// TIA Portal project "FinalPLC_V17" (V17)

(* hardware
DEVICE "S7-1200 station_1"  S7-1200 Station
   slot 0: "Rack_0"  S7-1200 Rack  Rack  V1.0
   slot 1: "PLC_1"  CPU 1211C DC/DC/DC  6ES7 211-1AE40-0XB0  V4.2
*)

// ===== PLC "PLC_1"  CPU 1211C DC/DC/DC =====

VAR_GLOBAL   // PLC tag table "Default tag table"
   "START" AT %I0.1 : Bool;
   "TG1" AT %M0.0 : Bool;
   "TG4" AT %M0.1 : Bool;
   "STOP" AT %I0.3 : Bool;
   "Emergency stop" AT %I0.4 : Bool;
   "AUTO" AT %I0.5 : Bool;
   "TG3" AT %M1.1 : Bool;
   "Entry Converyor" AT %Q0.0 : Bool;
   "Exit Converyor" AT %Q0.2 : Bool;
   "Start Light" AT %Q1.1 : Bool;
   "Start Light (Green)" AT %Q3.1 : Bool;
   "Stop Light (Red)" AT %Q3.3 : Bool;
   "Sensor 1" AT %I0.6 : Bool;
   "Vision sensor" AT %I0.0 : Bool;
   "Sensor 4" AT %I0.7 : Bool;
   "Output Vision" AT %ID30 : DInt;
   "Sortter 1 Turn" AT %Q0.3 : Bool;
   "TG STOP CG" AT %M0.2 : Bool;
   "Sortter 1 Belt" AT %Q0.4 : Bool;
   "RESET" AT %I0.2 : Bool;
   "Counter 1" AT %QD30 : DInt;
   "Sotter 2 Turn" AT %Q0.5 : Bool;
   "Sortter 2 Belt" AT %Q0.6 : Bool;
   "Counter 2" AT %QD34 : DInt;
   "Sotter 3 Turn" AT %Q0.7 : Bool;
   "Sotter 3 Belt" AT %Q1.0 : Bool;
   "Counter 3" AT %QD38 : DInt;
   "Counter 4" AT %QD42 : DInt;
   "TG5" AT %M0.5 : Bool;
   "Reset Light" AT %Q1.2 : Bool;
   "Reset Light (Yellow)" AT %Q3.2 : Bool;
   "Alarm Siren" AT %Q0.1 : Bool;
   "TG6" AT %M0.3 : Bool;
   "Grab 1" AT %Q2.3 : Bool;
   "Tag_1" AT %M100.0 : Bool;
   "Belt Converyor 1" AT %Q1.4 : Bool;
   "Belt Converyor 2" AT %Q1.5 : Bool;
   "Clamp 1" AT %Q1.7 : Bool;
   "Raise 1" AT %Q2.0 : Bool;
   "Sensor 3" AT %I1.1 : Bool;
   "Tag_2" AT %M100.1 : Bool;
   "Clamped 1" AT %I1.3 : Bool;
   "Mover Z1" AT %Q2.1 : Bool;
   "Detected 1" AT %I1.5 : Bool;
   "CB Sensor4" AT %M100.3 : Bool;
   "Moving Z1" AT %I1.6 : Bool;
   "Tag_10" AT %M101.1 : Bool;
   "Tag_3" AT %M100.2 : Bool;
   "Mover X1" AT %Q2.2 : Bool;
   "Clamp 2" AT %Q2.4 : Bool;
   "Clamped 2" AT %I2.0 : Bool;
   "Tag_5" AT %M100.4 : Bool;
   "Tag_6" AT %M100.5 : Bool;
   "Tag_8" AT %M100.7 : Bool;
   "Raise 2" AT %Q2.5 : Bool;
   "Tag_7" AT %M100.6 : Bool;
   "Sensor 2" AT %I1.0 : Bool;
   "Sensor box" AT %I1.2 : Bool;
   "Box converyor" AT %Q1.6 : Bool;
   "Tag_11" AT %M200.0 : Bool;
   "Mover Z2" AT %Q2.6 : Bool;
   "Mover X2" AT %Q2.7 : Bool;
   "Moving X2" AT %I2.4 : Bool;
   "Tag_12" AT %M200.1 : Bool;
   "Moving Z2" AT %I2.3 : Bool;
   "Tag_13" AT %M200.2 : Bool;
   "Grab 2" AT %Q3.0 : Bool;
   "Detected 2" AT %I2.2 : Bool;
   "Tag_14" AT %M200.3 : Bool;
   "Tag_15" AT %M200.4 : Bool;
   "Tag_19" AT %M200.7 : Bool;
   "Tag_16" AT %M200.5 : Bool;
   "Stop Light" AT %Q1.3 : Bool;
   "Tag_17" AT %M200.6 : Bool;
   "Tag_18" AT %QD46 : DInt;
   "Moving X1" AT %I1.7 : Bool;
   "Limit 1" AT %I1.4 : Bool;
   "TG2" AT %M1.0 : Bool;
   "MAN" AT %I2.5 : Bool;
   "IM_Con1" AT %I2.6 : Bool;
   "IM_Con2" AT %I2.7 : Bool;
   "IM_Con3" AT %I3.0 : Bool;
   "IM_Con4" AT %I3.1 : Bool;
   "IM_Alarm" AT %I3.2 : Bool;
END_VAR

// folder: System blocks/Program resources

DATA_BLOCK "IEC_Counter_0_DB"   // DB1
{ S7_Optimized_Access := 'TRUE' }
AUTHOR : SIMATIC
FAMILY : IEC
NAME : DCNTR
VERSION : 1.2
// stored: InstanceOfName IEC_DCOUNTER
"IEC_DCOUNTER"
BEGIN
END_DATA_BLOCK

DATA_BLOCK "IEC_Counter_0_DB_1"   // DB2
{ S7_Optimized_Access := 'TRUE' }
AUTHOR : SIMATIC
FAMILY : IEC
NAME : DCNTR
VERSION : 1.2
// stored: InstanceOfName IEC_DCOUNTER
"IEC_DCOUNTER"
BEGIN
END_DATA_BLOCK

DATA_BLOCK "IEC_Counter_0_DB_2"   // DB3
{ S7_Optimized_Access := 'TRUE' }
AUTHOR : SIMATIC
FAMILY : IEC
NAME : DCNTR
VERSION : 1.2
// stored: InstanceOfName IEC_DCOUNTER
"IEC_DCOUNTER"
BEGIN
END_DATA_BLOCK

DATA_BLOCK "IEC_Counter_0_DB_3"   // DB4
{ S7_Optimized_Access := 'TRUE' }
AUTHOR : SIMATIC
FAMILY : IEC
NAME : DCNTR
VERSION : 1.2
// stored: InstanceOfName IEC_DCOUNTER
"IEC_DCOUNTER"
BEGIN
END_DATA_BLOCK

DATA_BLOCK "IEC_Timer_0_DB"   // DB5
{ S7_Optimized_Access := 'TRUE' }
AUTHOR : Simatic
FAMILY : IEC
NAME : IEC_TMR
VERSION : 1.0
// stored: InstanceOfName IEC_TIMER
"IEC_TIMER"
BEGIN
END_DATA_BLOCK

DATA_BLOCK "IEC_Timer_0_DB_1"   // DB6
{ S7_Optimized_Access := 'TRUE' }
AUTHOR : Simatic
FAMILY : IEC
NAME : IEC_TMR
VERSION : 1.0
// stored: InstanceOfName IEC_TIMER
"IEC_TIMER"
BEGIN
END_DATA_BLOCK

DATA_BLOCK "IEC_Timer_0_DB_2"   // DB7
{ S7_Optimized_Access := 'TRUE' }
AUTHOR : Simatic
FAMILY : IEC
NAME : IEC_TMR
VERSION : 1.0
// stored: InstanceOfName IEC_TIMER
"IEC_TIMER"
BEGIN
END_DATA_BLOCK

DATA_BLOCK "IEC_Timer_0_DB_3"   // DB8
{ S7_Optimized_Access := 'TRUE' }
AUTHOR : Simatic
FAMILY : IEC
NAME : IEC_TMR
VERSION : 1.0
// stored: InstanceOfName IEC_TIMER
"IEC_TIMER"
BEGIN
END_DATA_BLOCK

DATA_BLOCK "IEC_Timer_0_DB_4"   // DB9
{ S7_Optimized_Access := 'TRUE' }
AUTHOR : Simatic
FAMILY : IEC
NAME : IEC_TMR
VERSION : 1.0
// stored: InstanceOfName IEC_TIMER
"IEC_TIMER"
BEGIN
END_DATA_BLOCK

DATA_BLOCK "IEC_Timer_0_DB_5"   // DB10
{ S7_Optimized_Access := 'TRUE' }
AUTHOR : Simatic
FAMILY : IEC
NAME : IEC_TMR
VERSION : 1.0
// stored: InstanceOfName IEC_TIMER
"IEC_TIMER"
BEGIN
END_DATA_BLOCK

DATA_BLOCK "IEC_Timer_0_DB_6"   // DB11
{ S7_Optimized_Access := 'TRUE' }
AUTHOR : Simatic
FAMILY : IEC
NAME : IEC_TMR
VERSION : 1.0
// stored: InstanceOfName IEC_TIMER
"IEC_TIMER"
BEGIN
END_DATA_BLOCK

DATA_BLOCK "IEC_Counter_0_DB_4"   // DB12
{ S7_Optimized_Access := 'TRUE' }
AUTHOR : SIMATIC
FAMILY : IEC
NAME : DCNTR
VERSION : 1.2
// stored: InstanceOfName IEC_DCOUNTER
"IEC_DCOUNTER"
BEGIN
END_DATA_BLOCK

// folder: (top level)

FUNCTION "Sorting station" : Void   // FC1, LAD
{ S7_Optimized_Access := 'TRUE' }
VERSION : 0.1
   VAR_TEMP   // added for the SCL form of the ladder/FBD networks
      _w1 : Bool;
   END_VAR
BEGIN

REGION Network 1: CHUONG TRINH
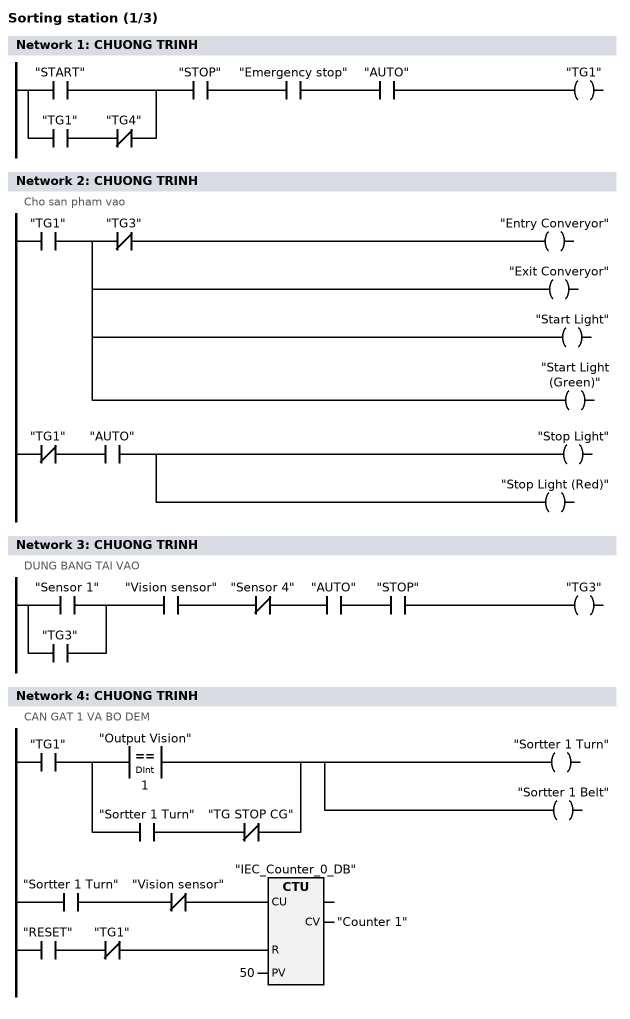
   RUNG wire#powerrail
      Contact( "START" )
      wire#w1
      Contact( "STOP" )
      Contact( "Emergency stop" )
      Contact( "AUTO" )
      Coil( "TG1" )
   END_RUNG
   RUNG wire#powerrail
      Contact( "TG1" )
      I_Contact( "TG4" )
   END_RUNG wire#w1
   // the same network as SCL:
   "TG1" := ("START" OR ("TG1" AND NOT "TG4")) AND "STOP" AND "Emergency stop" AND "AUTO";
END_REGION

REGION Network 2: CHUONG TRINH
   // Cho san pham vao
   RUNG wire#powerrail
      Contact( "TG1" )
      wire#w1
      I_Contact( "TG3" )
      Coil( "Entry Converyor" )
   END_RUNG
   RUNG wire#w1
      Coil( "Exit Converyor" )
   END_RUNG
   RUNG wire#w1
      Coil( "Start Light" )
   END_RUNG
   RUNG wire#w1
      Coil( "Start Light (Green)" )
   END_RUNG
   RUNG wire#powerrail
      I_Contact( "TG1" )
      Contact( "AUTO" )
      wire#w2
      Coil( "Stop Light" )
   END_RUNG
   RUNG wire#w2
      Coil( "Stop Light (Red)" )
   END_RUNG
   // the same network as SCL:
   "Entry Converyor" := "TG1" AND NOT "TG3";
   "Exit Converyor" := "TG1";
   "Start Light" := "TG1";
   "Start Light (Green)" := "TG1";
   "Stop Light" := NOT "TG1" AND "AUTO";
   "Stop Light (Red)" := "Stop Light";
END_REGION

REGION Network 3: CHUONG TRINH
   // DUNG BANG TAI VAO
   RUNG wire#powerrail
      Contact( "Sensor 1" )
      wire#w1
      Contact( "Vision sensor" )
      I_Contact( "Sensor 4" )
      Contact( "AUTO" )
      Contact( "STOP" )
      Coil( "TG3" )
   END_RUNG
   RUNG wire#powerrail
      Contact( "TG3" )
   END_RUNG wire#w1
   // the same network as SCL:
   "TG3" := ("Sensor 1" OR "TG3") AND "Vision sensor" AND NOT "Sensor 4" AND "AUTO" AND "STOP";
END_REGION

REGION Network 4: CHUONG TRINH
   // CAN GAT 1 VA BO DEM
   "Sortter 1 Turn" := "TG1" AND (("Output Vision" = 1) OR ("Sortter 1 Turn" AND NOT "TG STOP CG"));
   "Sortter 1 Belt" := "Sortter 1 Turn";
   "IEC_Counter_0_DB".CTU(CU := "Sortter 1 Turn" AND NOT "Vision sensor",
                          R := "RESET" AND NOT "TG1",
                          PV := 50,
                          CV => "Counter 1");
END_REGION

REGION Network 5: CHUONG TRINH
   // CAN GAT 2 VA BO DEM
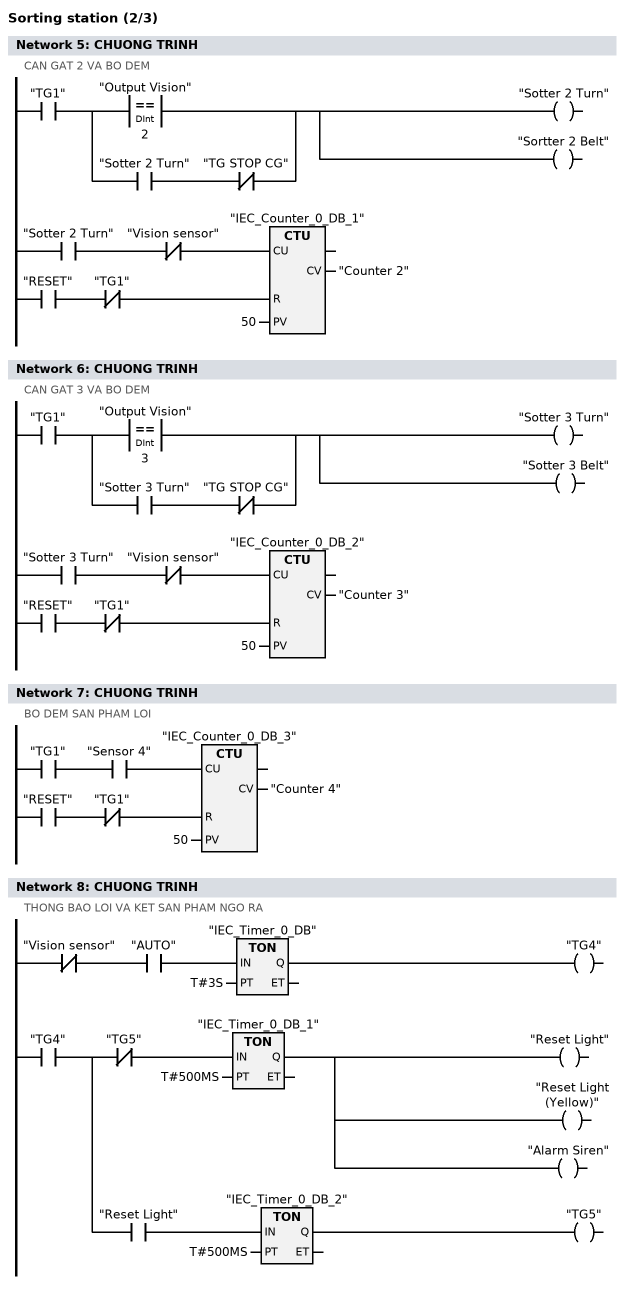
   "Sotter 2 Turn" := "TG1" AND (("Output Vision" = 2) OR ("Sotter 2 Turn" AND NOT "TG STOP CG"));
   "Sortter 2 Belt" := "Sotter 2 Turn";
   "IEC_Counter_0_DB_1".CTU(CU := "Sotter 2 Turn" AND NOT "Vision sensor",
                           R := "RESET" AND NOT "TG1",
                           PV := 50,
                           CV => "Counter 2");
END_REGION

REGION Network 6: CHUONG TRINH
   // CAN GAT 3 VA BO DEM
   "Sotter 3 Turn" := "TG1" AND (("Output Vision" = 3) OR ("Sotter 3 Turn" AND NOT "TG STOP CG"));
   "Sotter 3 Belt" := "Sotter 3 Turn";
   "IEC_Counter_0_DB_2".CTU(CU := "Sotter 3 Turn" AND NOT "Vision sensor",
                           R := "RESET" AND NOT "TG1",
                           PV := 50,
                           CV => "Counter 3");
END_REGION

REGION Network 7: CHUONG TRINH
   // BO DEM SAN PHAM LOI
   "IEC_Counter_0_DB_3".CTU(CU := "TG1" AND "Sensor 4", R := "RESET" AND NOT "TG1", PV := 50, CV => "Counter 4");
END_REGION

REGION Network 8: CHUONG TRINH
   // THONG BAO LOI VA KET SAN PHAM NGO RA
   "IEC_Timer_0_DB".TON(IN := NOT "Vision sensor" AND "AUTO", PT := T#3S);
   "TG4" := "IEC_Timer_0_DB".Q;
   "IEC_Timer_0_DB_1".TON(IN := "TG4" AND NOT "TG5", PT := T#500MS);
   "Reset Light" := "IEC_Timer_0_DB_1".Q;
   "Reset Light (Yellow)" := "IEC_Timer_0_DB_1".Q;
   "Alarm Siren" := "IEC_Timer_0_DB_1".Q;
   "IEC_Timer_0_DB_2".TON(IN := "TG4" AND "Reset Light", PT := T#500MS);
   "TG5" := "IEC_Timer_0_DB_2".Q;
END_REGION

REGION Network 9: CHUONG TRINH
   // THOI GIAN DELAY 1S CHO CAC CAN GAT
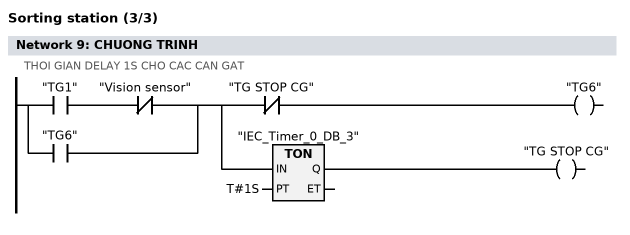
   #_w1 := ("TG1" AND NOT "Vision sensor") OR "TG6";
   "TG6" := #_w1 AND NOT "TG STOP CG";
   "IEC_Timer_0_DB_3".TON(IN := #_w1, PT := T#1S);
   "TG STOP CG" := "IEC_Timer_0_DB_3".Q;
END_REGION
END_FUNCTION

FUNCTION "Pick & Place 1" : Void   // FC2, LAD
{ S7_Optimized_Access := 'TRUE' }
VERSION : 0.1
   VAR_TEMP   // added for the SCL form of the ladder/FBD networks
      _w1 : Bool;
      _w2 : Bool;
      _w3 : Bool;
      _w4 : Bool;
      _w5 : Bool;
      _w6 : Bool;
   END_VAR
BEGIN

REGION Network 1
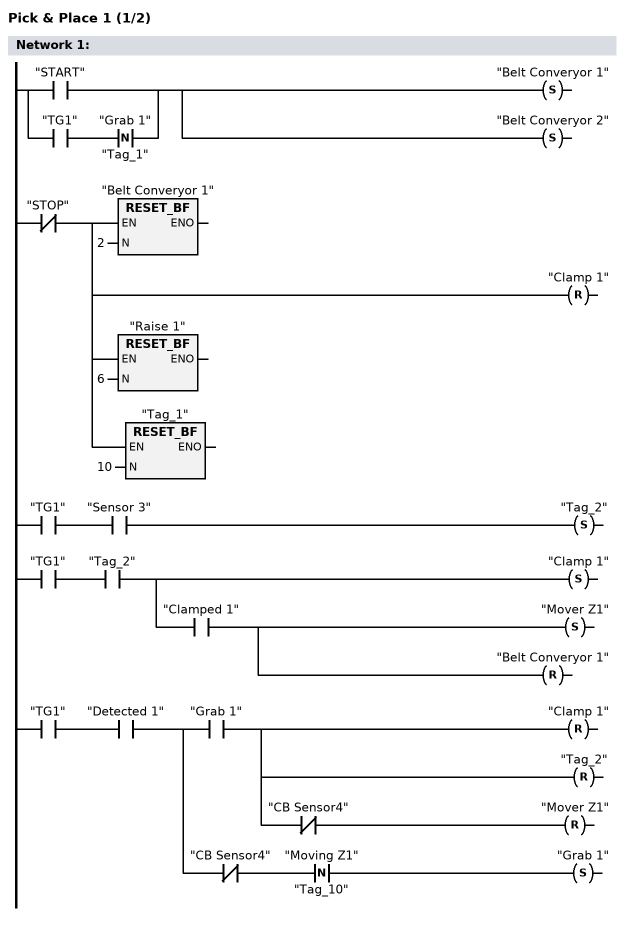
   // no SCL statement known for RBitfield: written as a call
   #_w1 := "TG1" AND NOT "Grab 1" AND "Tag_1";   // falling edge of "Grab 1"
   "Tag_1" := "Grab 1";
   IF "START" OR #_w1 THEN
       "Belt Converyor 1" := TRUE;
       "Belt Converyor 2" := TRUE;
   END_IF;
   #_w2 := NOT "STOP";
   IF #_w2 THEN
       RESET_BF(operand := "Belt Converyor 1", n := 2);
       "Clamp 1" := FALSE;
       RESET_BF(operand := "Raise 1", n := 6);
       RESET_BF(operand := "Tag_1", n := 10);
   END_IF;
   IF "TG1" AND "Sensor 3" THEN "Tag_2" := TRUE; END_IF;
   #_w3 := "TG1" AND "Tag_2";
   IF #_w3 THEN "Clamp 1" := TRUE; END_IF;
   IF #_w3 AND "Clamped 1" THEN
       "Mover Z1" := TRUE;
       "Belt Converyor 1" := FALSE;
   END_IF;
   #_w4 := "TG1" AND "Detected 1";
   #_w5 := #_w4 AND "Grab 1";
   IF #_w5 THEN
       "Clamp 1" := FALSE;
       "Tag_2" := FALSE;
   END_IF;
   IF #_w5 AND NOT "CB Sensor4" THEN "Mover Z1" := FALSE; END_IF;
   #_w6 := #_w4 AND NOT "CB Sensor4" AND NOT "Moving Z1" AND "Tag_10";   // falling edge of "Moving Z1"
   "Tag_10" := "Moving Z1";
   IF #_w6 THEN "Grab 1" := TRUE; END_IF;
END_REGION

REGION Network 2
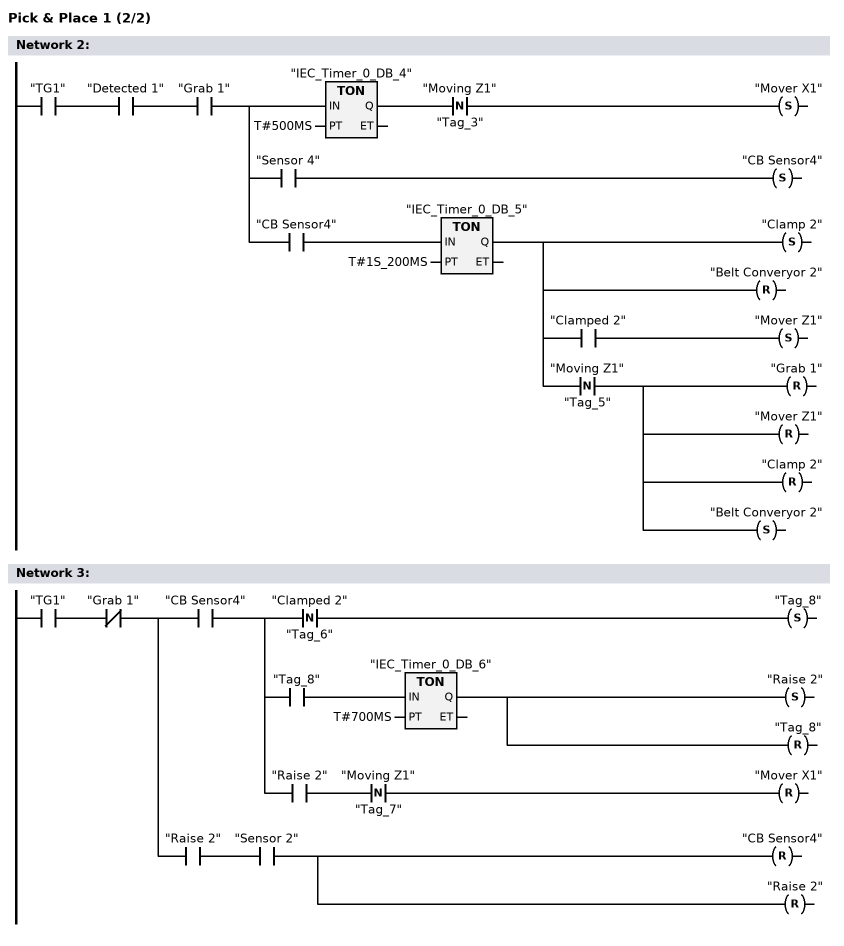
   #_w1 := "TG1" AND "Detected 1" AND "Grab 1";
   "IEC_Timer_0_DB_4".TON(IN := #_w1, PT := T#500MS);
   #_w2 := "IEC_Timer_0_DB_4".Q AND NOT "Moving Z1" AND "Tag_3";   // falling edge of "Moving Z1"
   "Tag_3" := "Moving Z1";
   IF #_w2 THEN "Mover X1" := TRUE; END_IF;
   IF #_w1 AND "Sensor 4" THEN "CB Sensor4" := TRUE; END_IF;
   "IEC_Timer_0_DB_5".TON(IN := #_w1 AND "CB Sensor4", PT := T#1S_200MS);
   IF "IEC_Timer_0_DB_5".Q THEN
       "Clamp 2" := TRUE;
       "Belt Converyor 2" := FALSE;
   END_IF;
   IF "IEC_Timer_0_DB_5".Q AND "Clamped 2" THEN "Mover Z1" := TRUE; END_IF;
   #_w3 := "IEC_Timer_0_DB_5".Q AND NOT "Moving Z1" AND "Tag_5";   // falling edge of "Moving Z1"
   "Tag_5" := "Moving Z1";
   IF #_w3 THEN
       "Grab 1" := FALSE;
       "Mover Z1" := FALSE;
       "Clamp 2" := FALSE;
       "Belt Converyor 2" := TRUE;
   END_IF;
END_REGION

REGION Network 3
   #_w1 := "TG1" AND NOT "Grab 1";
   #_w2 := #_w1 AND "CB Sensor4";
   #_w3 := #_w2 AND NOT "Clamped 2" AND "Tag_6";   // falling edge of "Clamped 2"
   "Tag_6" := "Clamped 2";
   IF #_w3 THEN "Tag_8" := TRUE; END_IF;
   "IEC_Timer_0_DB_6".TON(IN := #_w2 AND "Tag_8", PT := T#700MS);
   IF "IEC_Timer_0_DB_6".Q THEN
       "Raise 2" := TRUE;
       "Tag_8" := FALSE;
   END_IF;
   #_w4 := #_w2 AND "Raise 2" AND NOT "Moving Z1" AND "Tag_7";   // falling edge of "Moving Z1"
   "Tag_7" := "Moving Z1";
   IF #_w4 THEN "Mover X1" := FALSE; END_IF;
   IF #_w1 AND "Raise 2" AND "Sensor 2" THEN
       "CB Sensor4" := FALSE;
       "Raise 2" := FALSE;
   END_IF;
END_REGION
END_FUNCTION

FUNCTION "Pick & Place 2" : Void   // FC3, LAD
{ S7_Optimized_Access := 'TRUE' }
VERSION : 0.1
   VAR_TEMP   // added for the SCL form of the ladder/FBD networks
      _w1 : Bool;
      _w2 : Bool;
      _w3 : Bool;
      _w4 : Bool;
      _w5 : Bool;
      _w6 : Bool;
      _w7 : Bool;
      _w8 : Bool;
   END_VAR
BEGIN

REGION Network 1
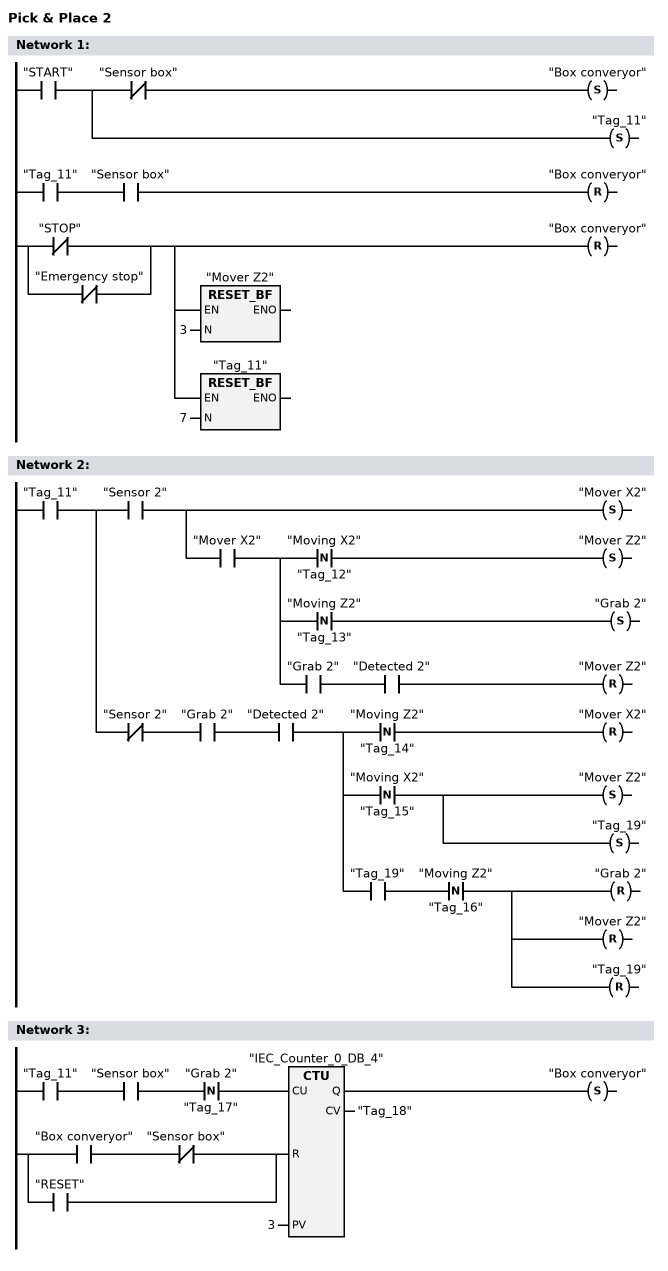
   // no SCL statement known for RBitfield: written as a call
   IF "START" AND NOT "Sensor box" THEN "Box converyor" := TRUE; END_IF;
   IF "START" THEN "Tag_11" := TRUE; END_IF;
   IF "Tag_11" AND "Sensor box" THEN "Box converyor" := FALSE; END_IF;
   IF NOT "STOP" OR NOT "Emergency stop" THEN "Box converyor" := FALSE; END_IF;
   #_w1 := NOT "STOP" OR NOT "Emergency stop";
   IF #_w1 THEN
       RESET_BF(operand := "Mover Z2", n := 3);
       RESET_BF(operand := "Tag_11", n := 7);
   END_IF;
END_REGION

REGION Network 2
   RUNG wire#powerrail
      Contact( "Tag_11" )
      wire#w1
      Contact( "Sensor 2" )
      wire#w2
      S_Coil( "Mover X2" )
   END_RUNG
   RUNG wire#w2
      Contact( "Mover X2" )
      wire#w3
      N_Contact(operand := "Moving X2", bit := "Tag_12")
      S_Coil( "Mover Z2" )
   END_RUNG
   RUNG wire#w3
      N_Contact(operand := "Moving Z2", bit := "Tag_13")
      S_Coil( "Grab 2" )
   END_RUNG
   RUNG wire#w3
      Contact( "Grab 2" )
      Contact( "Detected 2" )
      R_Coil( "Mover Z2" )
   END_RUNG
   RUNG wire#w1
      I_Contact( "Sensor 2" )
      Contact( "Grab 2" )
      Contact( "Detected 2" )
      wire#w4
      N_Contact(operand := "Moving Z2", bit := "Tag_14")
      R_Coil( "Mover X2" )
   END_RUNG
   RUNG wire#w4
      N_Contact(operand := "Moving X2", bit := "Tag_15")
      wire#w5
      S_Coil( "Mover Z2" )
   END_RUNG
   RUNG wire#w5
      S_Coil( "Tag_19" )
   END_RUNG
   RUNG wire#w4
      Contact( "Tag_19" )
      N_Contact(operand := "Moving Z2", bit := "Tag_16")
      wire#w6
      R_Coil( "Grab 2" )
   END_RUNG
   RUNG wire#w6
      R_Coil( "Mover Z2" )
   END_RUNG
   RUNG wire#w6
      R_Coil( "Tag_19" )
   END_RUNG
   // the same network as SCL:
   #_w1 := "Tag_11" AND "Sensor 2";
   IF #_w1 THEN "Mover X2" := TRUE; END_IF;
   #_w2 := #_w1 AND "Mover X2";
   #_w3 := #_w2 AND NOT "Moving X2" AND "Tag_12";   // falling edge of "Moving X2"
   "Tag_12" := "Moving X2";
   IF #_w3 THEN "Mover Z2" := TRUE; END_IF;
   #_w4 := #_w2 AND NOT "Moving Z2" AND "Tag_13";   // falling edge of "Moving Z2"
   "Tag_13" := "Moving Z2";
   IF #_w4 THEN "Grab 2" := TRUE; END_IF;
   IF #_w2 AND "Grab 2" AND "Detected 2" THEN "Mover Z2" := FALSE; END_IF;
   #_w5 := "Tag_11" AND NOT "Sensor 2" AND "Grab 2" AND "Detected 2";
   #_w6 := #_w5 AND NOT "Moving Z2" AND "Tag_14";   // falling edge of "Moving Z2"
   "Tag_14" := "Moving Z2";
   IF #_w6 THEN "Mover X2" := FALSE; END_IF;
   #_w7 := #_w5 AND NOT "Moving X2" AND "Tag_15";   // falling edge of "Moving X2"
   "Tag_15" := "Moving X2";
   IF #_w7 THEN
       "Mover Z2" := TRUE;
       "Tag_19" := TRUE;
   END_IF;
   #_w8 := #_w5 AND "Tag_19" AND NOT "Moving Z2" AND "Tag_16";   // falling edge of "Moving Z2"
   "Tag_16" := "Moving Z2";
   IF #_w8 THEN
       "Grab 2" := FALSE;
       "Mover Z2" := FALSE;
       "Tag_19" := FALSE;
   END_IF;
END_REGION

REGION Network 3
   #_w1 := "Tag_11" AND "Sensor box" AND NOT "Grab 2" AND "Tag_17";   // falling edge of "Grab 2"
   "Tag_17" := "Grab 2";
   "IEC_Counter_0_DB_4".CTU(CU := #_w1,
                           R := ("Box converyor" AND NOT "Sensor box") OR "RESET",
                           PV := 3,
                           CV => "Tag_18");
   IF "IEC_Counter_0_DB_4".Q THEN "Box converyor" := TRUE; END_IF;
END_REGION
END_FUNCTION

FUNCTION "Manual" : Void   // FC4, LAD
{ S7_Optimized_Access := 'TRUE' }
VERSION : 0.1
BEGIN

REGION Network 1
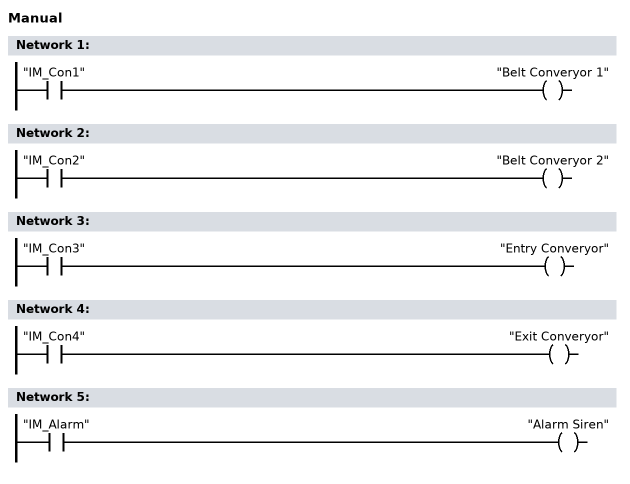
   RUNG wire#powerrail
      Contact( "IM_Con1" )
      Coil( "Belt Converyor 1" )
   END_RUNG
   // the same network as SCL:
   "Belt Converyor 1" := "IM_Con1";
END_REGION

REGION Network 2
   RUNG wire#powerrail
      Contact( "IM_Con2" )
      Coil( "Belt Converyor 2" )
   END_RUNG
   // the same network as SCL:
   "Belt Converyor 2" := "IM_Con2";
END_REGION

REGION Network 3
   RUNG wire#powerrail
      Contact( "IM_Con3" )
      Coil( "Entry Converyor" )
   END_RUNG
   // the same network as SCL:
   "Entry Converyor" := "IM_Con3";
END_REGION

REGION Network 4
   RUNG wire#powerrail
      Contact( "IM_Con4" )
      Coil( "Exit Converyor" )
   END_RUNG
   // the same network as SCL:
   "Exit Converyor" := "IM_Con4";
END_REGION

REGION Network 5
   RUNG wire#powerrail
      Contact( "IM_Alarm" )
      Coil( "Alarm Siren" )
   END_RUNG
   // the same network as SCL:
   "Alarm Siren" := "IM_Alarm";
END_REGION
END_FUNCTION

FUNCTION "MHJ-PLC-Lab-Function-S71200" : Void   // FC9000, SCL
{ S7_Optimized_Access := 'TRUE' }
VERSION : 0.1
   VAR_TEMP
      rdTimeReturn : Int;
      outputTime : DTL;
      SyncVal : Byte;
      forVal : Int;
      forVal_2 : Int;
      Value : Byte;
   END_VAR
   VAR CONSTANT
      CompVal : Byte := 16#34;
      Value_01 : Byte := 16#11;
      Value_01_DW : DWord := 16#A165_D992;
      Value_02_DW : DWord := 16#58BE_4401;
   END_VAR
BEGIN

   #Value:=PEEK(area := 16#82,
        dbNumber := 0,
        byteOffset := 511);
   #Value := #Value + 1;

   POKE(area := 16#82,
        dbNumber := 0,
        byteOffset := 511,
        value := #Value);

   POKE(area:=16#81,
        dbNumber:=0,
        byteOffset:=1016,
        value:=#Value_01_DW);
   POKE(area := 16#81,
        dbNumber := 0,
        byteOffset := 1020,
        value := #Value_02_DW);

   POKE(area := 16#81,
        dbNumber := 0,
        byteOffset := 511,
        value := B#16#00);

   FOR #forVal := 0 TO 120 DO
       FOR #forVal_2:=0 TO 10 DO
           #rdTimeReturn:=RD_SYS_T(#outputTime);
           #rdTimeReturn := WR_SYS_T(#outputTime);
           #rdTimeReturn := RD_SYS_T(#outputTime);
           #rdTimeReturn := WR_SYS_T(#outputTime);
       END_FOR;
       #SyncVal:= PEEK(area := 16#81,
                      dbNumber := 0,
                      byteOffset := 511);
       IF #SyncVal = #CompVal THEN
          GOTO M_1;
       END_IF;
   END_FOR;
   RETURN;

   M_1:
   POKE(area := 16#81,
        dbNumber := 0,
        byteOffset := 511,
        value := B#16#0);
END_FUNCTION

ORGANIZATION_BLOCK "Main"   // OB1, LAD, ProgramCycle
TITLE = "Main Program Sweep (Cycle)"
{ S7_Optimized_Access := 'TRUE' }
VERSION : 0.1
   VAR_INPUT
      Initial_Call : Bool;   // Initial call of this OB
      Remanence : Bool;   // =True, if remanent data are available
   END_VAR
BEGIN

REGION Network 1
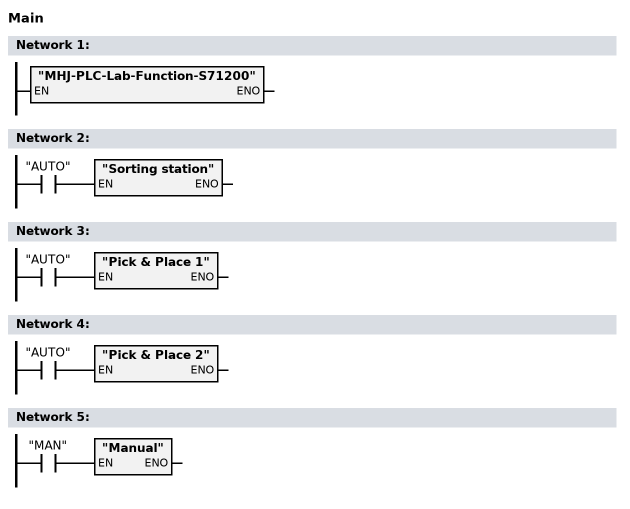
   RUNG wire#powerrail
      "MHJ-PLC-Lab-Function-S71200"()
   END_RUNG
   // the same network as SCL:
   "MHJ-PLC-Lab-Function-S71200"();
END_REGION

REGION Network 2
   RUNG wire#powerrail
      Contact( "AUTO" )
      "Sorting station"()
   END_RUNG
   // the same network as SCL:
   IF "AUTO" THEN "Sorting station"(); END_IF;
END_REGION

REGION Network 3
   RUNG wire#powerrail
      Contact( "AUTO" )
      "Pick & Place 1"()
   END_RUNG
   // the same network as SCL:
   IF "AUTO" THEN "Pick & Place 1"(); END_IF;
END_REGION

REGION Network 4
   RUNG wire#powerrail
      Contact( "AUTO" )
      "Pick & Place 2"()
   END_RUNG
   // the same network as SCL:
   IF "AUTO" THEN "Pick & Place 2"(); END_IF;
END_REGION

REGION Network 5
   RUNG wire#powerrail
      Contact( "MAN" )
      "Manual"()
   END_RUNG
   // the same network as SCL:
   IF "MAN" THEN "Manual"(); END_IF;
END_REGION
END_ORGANIZATION_BLOCK